{attribute 'GeneratedUsingTerminal: EP9224-0037-0017'}
{attribute addProperty BoxType "EP9224-0037-0017"}
{attribute addProperty Id "Error_UsBOOL1Error_UpBOOL1Warning_UsBOOL1Warning_UpBOOL1Status_UsBOOL1Status_UpBOOL1Channel_ErrorBOOL1Error_Sum_CurrentBOOL1Warning_Sum_CurrentBOOL1TxPDO_StateBOOL1TxPDO_ToggleBOOL1"}
{attribute addProperty CRC "363647489"}
{attribute addProperty Size "11"}
TYPE Status_15ACD201 :
STRUCT
	{attribute addProperty Name "Error_Us"}
	Error_Us : BOOL;
	{attribute addProperty Name "Error_Up"}
	Error_Up : BOOL;
	{attribute addProperty Name "Warning_Us"}
	Warning_Us : BOOL;
	{attribute addProperty Name "Warning_Up"}
	Warning_Up : BOOL;
	{attribute addProperty Name "Status_Us"}
	Status_Us : BOOL;
	{attribute addProperty Name "Status_Up"}
	Status_Up : BOOL;
	{attribute addProperty Name "Channel_Error"}
	Channel_Error : BOOL;
	{attribute addProperty Name "Error_Sum_Current"}
	Error_Sum_Current : BOOL;
	{attribute addProperty Name "Warning_Sum_Current"}
	Warning_Sum_Current : BOOL;
	{attribute addProperty Name "TxPDO_State"}
	TxPDO_State : BOOL;
	{attribute addProperty Name "TxPDO_Toggle"}
	TxPDO_Toggle : BOOL;
END_STRUCT
END_TYPE

(* stored: Version 1.2.0.0, ProductVersion 3.1.4024.9
   DUT Status_15ACD201: Id {91a5cfed-c946-4ad8-bf0d-2b155782cf46} *)
